FUNCTION F_PB_GetTuDestination : E_FunctionNumber
VAR_INPUT
	eFunctionNumber		: E_FunctionNumber; // Function number
	ZoneNumber			: INT; // ZoneNumber
	TuTableDestIdx		: INT; // Which Tu Table destination slot (Default 1)
END_VAR
VAR_OUTPUT	
	TU_DataIndex		: DINT;
END_VAR


IF( ZoneNumber > 0 AND ZoneNumber <= Conveyor.NUMBER_OF_ZONES_PER_FUNCTION) THEN

		// If zone is valid and consists of a TU-Data index
		IF __ISVALIDREF(FunctionRegistry[eFunctionNumber].Zone[ZoneNumber].refZoneData) THEN
			TU_DataIndex := FunctionRegistry[eFunctionNumber].Zone[ZoneNumber].refZoneData.TransportControlData.TU_DataIndex;
			 IF TU_DataIndex > 0 THEN
				// Return destination slot
				F_PB_GetTuDestination := TU_DataTable[TU_DataIndex].Destination[TuTableDestIdx].eFunctionNumber;				
			 END_IF
		END_IF	
END_IF

END_FUNCTION

(* stored: Version 1.1.0.1, ProductVersion 3.1.4024.9
   POU F_PB_GetTuDestination: Id {67064ea1-6b0d-42c1-b28a-a11d48c498a1}, SpecialFunc None *)
